TYPE ST_AteqRecipe :
STRUCT
	bEnabled : BOOL;
	nNumOfActivePrograms	: UINT;
END_STRUCT
END_TYPE

(* stored: Version 1.1.0.1
   DUT ST_AteqRecipe: Id {ee45e8df-e534-0732-329b-2d34692732d3} *)
